FUNCTION_BLOCK INTEGRAL_REAL
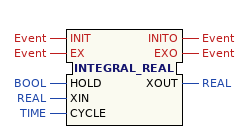
  EVENT_INPUT
    INIT;
    EX;
  END_EVENT
  EVENT_OUTPUT
    INITO;
    EXO;
  END_EVENT
  VAR_INPUT
    HOLD : BOOL;
    XIN : REAL;
    CYCLE : TIME;
  END_VAR
  VAR_OUTPUT
    XOUT : REAL;
  END_VAR
  EC_STATES
    START;
  END_STATES
END_FUNCTION_BLOCK
